FUNCTION_BLOCK ListOfUserDatatype EXTENDS WrappableList
VAR_INPUT
END_VAR
VAR_OUTPUT
END_VAR
VAR
END_VAR

METHOD Append : REFERENCE TO ListOfUserDatatype
VAR_INPUT
	data : UserDatatype;
END_VAR
Append REF= THIS^;
SUPER^._Append(data);
END_METHOD


METHOD Get : REFERENCE TO UserDatatype
VAR_INPUT
	index : INT;
END_VAR
VAR
	value : UserDatatype;
END_VAR

_Get(index, value);
Get REF= value;
END_METHOD

END_FUNCTION_BLOCK

(* stored: Version 1.1.0.1, ProductVersion 3.1.4024.11
   POU ListOfUserDatatype: Id {8aeba194-e122-497c-bdbb-6b4adc25f2d1}, SpecialFunc None
   Method Append: Id {7fa7eaa6-6436-44e9-9d7b-b083be30978c}
   Method Get: Id {53990a68-dd1b-4daa-a571-3a5dca3db2e6} *)
